# EPICS substitutions: db/Beckhoff_9XXX/ecmcEL9505.substitutions
file "ecmcEcSlave.template"
{
  pattern {}
          {}
}

file "ecmcEL95XX-chX.template"
{
  pattern {CH_ID}
          {01   }
}
